(*
SPDX-FileCopyrightText: © 2026 Oleksandr Tiutyk <trofimich@gmail.com>
SPDX-License-Identifier: MIT
License: https://opensource.org/license/mit
*)

INTERFACE IArgumentValueNotSupportedException EXTENDS IGeneralException

METHOD Throw
VAR_INPUT
	sourceNamespaceName : STRING;
	sourceClassName : STRING;
	sourcePOUName : STRING;
	sourcePosition : STRING;
	argumentName : STRING;
	argumentValue : ANY;
END_VAR
END_METHOD

END_INTERFACE

(* stored: Version 1.1.0.1
   Itf IArgumentValueNotSupportedException: Id {8874df74-44d8-499c-99ad-cd9b0f0621ad}
   Method Throw: Id {b95db194-afbb-41f7-9a2a-484dfac8ba09} *)
